(* IEC 61131-3 sources: CodesysTest/alpha/export/FBs/Components/Aux IO/FB_AuxIOPhysical.pou, 3 files *)

(* ---- FB_AuxIOPhysical.pou.st ---- *)
(*#-#-#-#-#-#-#-#-#-#---Declaration---#-#-#-#-#-#-#-#-#-#-#-#-#*)

FUNCTION_BLOCK FINAL FB_AuxIOPhysical
VAR_INPUT
	bagsLow : BOOL;
	configIn1 : BOOL;
	configIn2 : BOOL;
	configIn3 : BOOL;
	configIn4 : BOOL;
	faultActive : BOOL;
	inhibitCycle : BOOL;
	printerDataReady : BOOL;
	waitingForFiller : BOOL;
	runExitConveyor : BOOL;
	state : StateMachine;
	factorySelection : AuxIOConfiguration;
	fillerType : REFERENCE TO FillerSelection;
END_VAR
VAR_OUTPUT
	baggerOK : BOOL;
	fillerOK : BOOL;
	configOut1 : BOOL;
	configOut2 : BOOL;
	bagGrabbed : BOOL;
	inhibitBagger : BOOL;
	reverseConveyor : BOOL;
	readyForFiller : BOOL;
	collisionDetected : BOOL;
END_VAR
VAR
	_configOutputManager : FB_OutputPulseManager;
	_outputPulse_CycleComplete : FB_MonostableMultivibrator();
	_OutputPulse_BagMade : FB_MonostableMultivibrator();
	_heartbeatWarningTimerOn : TON := (PT := T#1000MS);
	_heartbeatWarningTimerOff : TON := (PT := T#1000MS);
	_readyForGrab : BOOL;
	_readyForGrabONS : Standard.R_TRIG();
END_VAR

(*#-#-#-#-#-#-#-#-#-#---Implementation---#-#-#-#-#-#-#-#-#-#-#-#-#*)

//
_configOutputManager();

//
CASE factorySelection.factorySelection OF
    AuxiliaryIOSelection.NotInstalled:
    //

    AuxiliaryIOSelection.AuxIOStandard:

        (* Outputs of AuxIO Block *)

        // Baggers not faults and heated up.
        baggerOK := NOT faultActive;

        // Bags open and ready for filler.
        readyForFiller := waitingForFiller;

        // Active if either input is set to 'FillerOK' and the corresponding input is active.
        fillerOK := InputActive(AuxInputSelection.FillerOK);

        // Active if either input is set to 'BaggerInhibit' and the corresponding input is active, or PAA enabled and inhibiting cycle.
        inhibitBagger := InputActive(AuxInputSelection.BaggerInhibit) OR inhibitCycle;

		// Optional Collision Detection on config input
		collisionDetected := InputActive(AuxInputSelection.CollisionDetection);

        // Custom PRJ-22085: Robot successfully grabbed bag.
        bagGrabbed := InputActive(AuxInputSelection.BagGrabbed);

        // Custom PRJ-59126: Reverse BEC when high
        reverseConveyor := InputActive(AuxInputSelection.ReverseConveyor);

        (* Configurable Outputs *)

        // Custom PRJ22085: Ready For Grab
        _readyForGrabONS(CLK := waitingForFiller);

        IF _readyForGrabONS.Q THEN
            SetReadyForGrab();
        END_IF

        IF _readyForGrab THEN
            _configOutputManager.ManualOn(OutputSelected(AuxOutputSelection.ReadyForGrab));
        ELSE
            _configOutputManager.ManualOff(OutputSelected(AuxOutputSelection.ReadyForGrab));
        END_IF

        // Bags Low
        IF bagsLow THEN
            _configOutputManager.ManualOn(OutputSelected(AuxOutputSelection.BagsLow));
        ELSE
            _configOutputManager.ManualOff(OutputSelected(AuxOutputSelection.BagsLow));
        END_IF

        // Cycle Complete
        IF state.head = HEAD_STATES.OpenedBag THEN
            _configOutputManager.Trigger(OutputSelected(AuxOutputSelection.CycleComplete));
        END_IF

        // Bag Made
        IF state.head = HEAD_STATES.SealedAndSeparatedBag THEN
            _configOutputManager.Trigger(OutputSelected(AuxOutputSelection.BagMade));
        END_IF

        // Printer Data Ready
        IF printerDataReady THEN
            _configOutputManager.ManualOn(OutputSelected(AuxOutputSelection.PrinterDataReady));
        ELSE
            _configOutputManager.ManualOff(OutputSelected(AuxOutputSelection.PrinterDataReady));
        END_IF

        // Waiting For Printer
        IF state.sb.releaseFeed = RELEASE_FEED_STATES.WaitForPrinter THEN
            _configOutputManager.ManualOn(OutputSelected(AuxOutputSelection.WaitingForPrinter));
        ELSE
            _configOutputManager.ManualOff(OutputSelected(AuxOutputSelection.WaitingForPrinter));
        END_IF

        // Bag Made Plus Label Required
        IF NOT printerDataReady AND state.head = HEAD_STATES.SealedAndSeparatedBag THEN
            _configOutputManager.ManualOn(OutputSelected(AuxOutputSelection.BagMadePlusLabelRequired));
        END_IF

        IF printerDataReady OR faultActive OR (state.sb.releaseFeed = RELEASE_FEED_STATES.FeedToOffset) THEN
            _configOutputManager.ManualOff(OutputSelected(AuxOutputSelection.BagMadePlusLabelRequired));
        END_IF

        // Exit Conveyor
        IF runExitConveyor THEN
            _configOutputManager.ManualOn(OutputSelected(AuxOutputSelection.RunExternalExitConveyor));
        ELSE
            _configOutputManager.ManualOff(OutputSelected(AuxOutputSelection.RunExternalExitConveyor));
        END_IF

        configOut1 := _configOutputManager.configOut1;
        configOut2 := _configOutputManager.configOut2;
END_CASE

(* ---- Reset.m.st ---- *)
(*#-#-#-#-#-#-#-#-#-#---Declaration---#-#-#-#-#-#-#-#-#-#-#-#-#*)

METHOD Reset
VAR_INPUT
END_VAR
(*#-#-#-#-#-#-#-#-#-#---Implementation---#-#-#-#-#-#-#-#-#-#-#-#-#*)

_configOutputManager.reset();
_readyForGrab := FALSE;

(* ---- SetReadyForGrab.m.st ---- *)
(*#-#-#-#-#-#-#-#-#-#---Declaration---#-#-#-#-#-#-#-#-#-#-#-#-#*)

METHOD SetReadyForGrab : BOOL
VAR_INPUT
END_VAR
(*#-#-#-#-#-#-#-#-#-#---Implementation---#-#-#-#-#-#-#-#-#-#-#-#-#*)

_readyForGrab := TRUE;
